FUNCTION F_LogError : STRING;
VAR_INPUT
	Message : T_MaxString;
END_VAR

F_LogError := F_Logger(ADSLOG_MSGTYPE_ERROR, Message);

END_FUNCTION

(* stored: Version 1.1.0.1, ProductVersion 3.1.4020.12
   POU F_LogError: Id {66d67573-6e40-4463-a296-d64414f9bf59}, SpecialFunc None *)
